// TwinCAT 3 PLC project main
// ProgramVersion: 3.1.4024.0
// libraries:
//   Tc2_Standard, * (Beckhoff Automation GmbH)
//   Tc2_System, * (Beckhoff Automation GmbH)
//   Tc3_Module, * (Beckhoff Automation GmbH)
// project tree:
//   / GlobalTextList.TcGTLO, PlcTask.TcTTO, Visualization Manager.TcVMO (not stored)
//   POUs/ MAIN.TcPOU
//   VISUs/ Visu.TcVIS

CONFIGURATION main
    RESOURCE PLC ON TwinCAT3
        TASK PlcTask(INTERVAL := T#10ms, PRIORITY := 20);
        PROGRAM MAIN WITH PlcTask : MAIN;
    END_RESOURCE
END_CONFIGURATION

// ---- POUs/MAIN.TcPOU
PROGRAM MAIN
VAR
	bS1 	: BOOL; //Sensor hoog niveau
	bS2 	: BOOL; //Sensor laag niveau
	bK1 	: BOOL; //Klep
	bP1 	: BOOL; //Pomp
	bStart 	: BOOL; //Start de pomp
	bStop 	: BOOL; //Stop de pomp
END_VAR

//Een opslagvat heeft twee sensoren in de zijwand die een laag en hoog niveau aanduiden. 
//Aan de hand van een PLC programma dient er automatisch de klep bovenaan het vat geopend te worden als het vat leeg is. 
//De tank wordt nu gevuld. Als de tank vol is sluit de klep K1 eveneens automatisch. 
//Onderaan de tank bevindt zich een pomp P1 die met een start- en stop-drukknop in- en uitgeschakeld kan worden. 

//Als de tank leeg gelopen is, stopt de pomp automatisch en opent de klep K1 bovenaan. 
//De pomp kan niet ingeschakeld worden zolang de tank gevuld wordt.

//bS1 detecteert geen vloeistof -> false
//bS2 detecteert geen vloeistof -> false
//bK1 is open -> true
//bP1 is aan -> ture

bK1 := NOT bS1 AND NOT bS2;
bP1 := NOT bStop AND bStart AND NOT bS2;
IF bStop THEN
	bStart := FALSE;
END_IF

IF bK1 THEN
	bP1 :=  FALSE;
END_IF

END_PROGRAM

// ---- GlobalTextList.TcGTLO
TEXTLIST GlobalTextList
  200 = 'bK1'
  201 = 'bP1'
  16 = 'bS1'
  784 = 'bS2'
  586 = 'bStart'
  609 = 'bStop'
END_TEXTLIST

// ---- VISUs/Visu.TcVIS
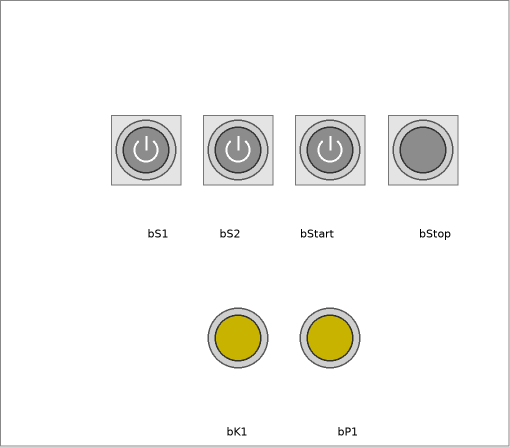
VISUALIZATION Visu  // 510x447
    PowerSwitch (111,115 70x70), variable: MAIN.bS1, behaviour: TOGGLE, style: Switch-PowerSwitch-Gray
    PowerSwitch (203,115 70x70), variable: MAIN.bS2, behaviour: TOGGLE, style: Switch-PowerSwitch-Gray
    PowerSwitch (295,115 70x70), variable: MAIN.bStart, behaviour: TOGGLE, style: Switch-PowerSwitch-Gray
    PushSwitch (388,115 70x70), variable: MAIN.bStop, behaviour: TOGGLE, style: Switch-PushSwitch-Gray
    Lamp1 (203,303 70x70), variable: MAIN.bK1, style: Lamp-Lamp1-Yellow
    Lamp1 (295,303 70x70), variable: MAIN.bP1, style: Lamp-Lamp1-Yellow
    Label (83,219 150x30), "bS1"
    Label (155,219 150x30), "bS2"
    Label (242,219 150x30), "bStart"
    Label (360,219 150x30), "bStop"
    Label (162,417 150x30), "bK1"
    Label (273,417 150x30), "bP1"
END_VISUALIZATION
